FUNCTION F_NOW (* returns current local date and time *)
  PACKAGE eclipse4diac::utils::timing;
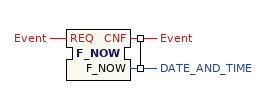
  EVENT_INPUT
    REQ;
  END_EVENT
  EVENT_OUTPUT
    CNF WITH F_NOW;
  END_EVENT
  VAR_OUTPUT
    F_NOW : DATE_AND_TIME;
  END_VAR
  BODY IN ST:
PACKAGE utils::timing;

(* returns current local date and time *)
FUNCTION F_NOW : DATE_AND_TIME
F_NOW := NOW();
END_FUNCTION
  END_BODY
END_FUNCTION
